TYPE ST_System_AKM_Parameter :
STRUCT

	Zeit_Nachl						: REAL;
	Zeit_Vorl							: REAL;

	AutoQuittierung					: BOOL;

	Stellwert_Temperatur_KW_Max		: REAL;
	Stellwert_Temperatur_KW_Min		: REAL;
	Stellwert_Temperatur_WW_Max		: REAL;
	Stellwert_Temperatur_WW_Min		: REAL;

	Temp_Heisswasser		        : REAL;
	Temp_Heisswasser_Max	        : REAL;
	Temp_Heisswasser_Min	        : REAL;

	Temp_Warmwasser			        : REAL;
	Temp_Warmwasser_Max		        : REAL;
	Temp_Warmwasser_Min		        : REAL;

	Temp_Kaltwasser			        : REAL;
	Temp_Kaltwasser_Max		        : REAL;
	Temp_Kaltwasser_Min		        : REAL;


END_STRUCT
END_TYPE

(* stored: Version 1.1.0.1, ProductVersion 3.1.4024.9
   DUT ST_System_AKM_Parameter: Id {62a39cf8-9317-4fcd-a4fd-a4b59bc68feb} *)
